FUNCTION_BLOCK ScrollFS_PHYS_Button (* Scroll list — accepts a single ScrollFull_S struct (geometry + physical controls), reads 6 on-screen Buttons and the direct-position input field, drives ScrollFS internally *)
  (* Standard: ISO 11783-6; Description: Copyright (c) 2026 Meisterschulen am Ostbahnhof This program and the accompanying materials are made available under the terms of the Eclipse Public License 2.0 which is available at https://www.eclipse.org/legal/epl-2.0/ SPDX-License-Identifier: EPL-2.0 Same as ScrollFS_PHYS, but reads the 6 scroll controls as on-screen Button objects (Button_IE, listening for BT_PRESSED_LATCHED) instead of physical SoftKeys — for masks where scrolling is operated via touch/on-screen buttons rather than the SoftKey column. Reuses the same ScrollFull_S / ScrollControls_S structs (the 6 IDs just point at Button objects instead of Key objects) and the same internal ScrollFS position engine. See Workspace_Scroll/SCROLL_KONZEPT.md for the full derivation. *)
  (* Version 1.1, 2026-09-05, Franz Höpfinger, Meisterschulen am Ostbahnhof, Add xScale flag, passed through to the internal ScrollFS *)
  (* Version 1.0, 2026-08-09, Franz Höpfinger, Meisterschulen am Ostbahnhof, initial API and implementation and/or initial documentation *)
  PACKAGE isobus::UT::Q;
  IMPORT isobus::utils::scroll::ScrollFull_S;
  IMPORT isobus::UT::Q::ScrollFS;
  IMPORT iec61131::selection::F_MOVE;
  IMPORT iec61131::conversion::F_DWORD_TO_DINT;
  IMPORT isobus::UT::io::Button::Button_IE;
  IMPORT isobus::UT::io::Button::ButtonActivationCode::BT_PRESSED_LATCHED;
  IMPORT isobus::UT::io::NumericValue::NumericValue_ID;
  IMPORT isobus::UT::Q::Q_NumericValue;
  IMPORT isobus::UT::Q::const::IDs::ID_NULL;
  IMPORT iec61131::selection::F_SEL;
  IMPORT iec61131::conversion::F_UINT_TO_UDINT;
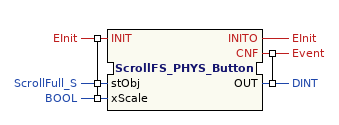
  EVENT_INPUT
    INIT : EInit WITH stObj, xScale; (* Service Initialization *)
  END_EVENT
  EVENT_OUTPUT
    INITO : EInit; (* Initialization Confirm *)
    CNF WITH OUT; (* Confirmation of a position change *)
  END_EVENT
  VAR_INPUT
    stObj : isobus::utils::scroll::ScrollFull_S; (* Complete scroll list configuration (geometry + operator controls), snapshotted at INIT *)
    xScale : BOOL := FALSE; (* FALSE (default) = bypass. TRUE = scale by the DM/SKM factor. Passed straight through to the internal ScrollFS instance. *)
  END_VAR
  VAR_OUTPUT
    OUT : DINT; (* Current scroll position (0..stObj.stGeometry.i32PosMax, in rows) *)
  END_VAR
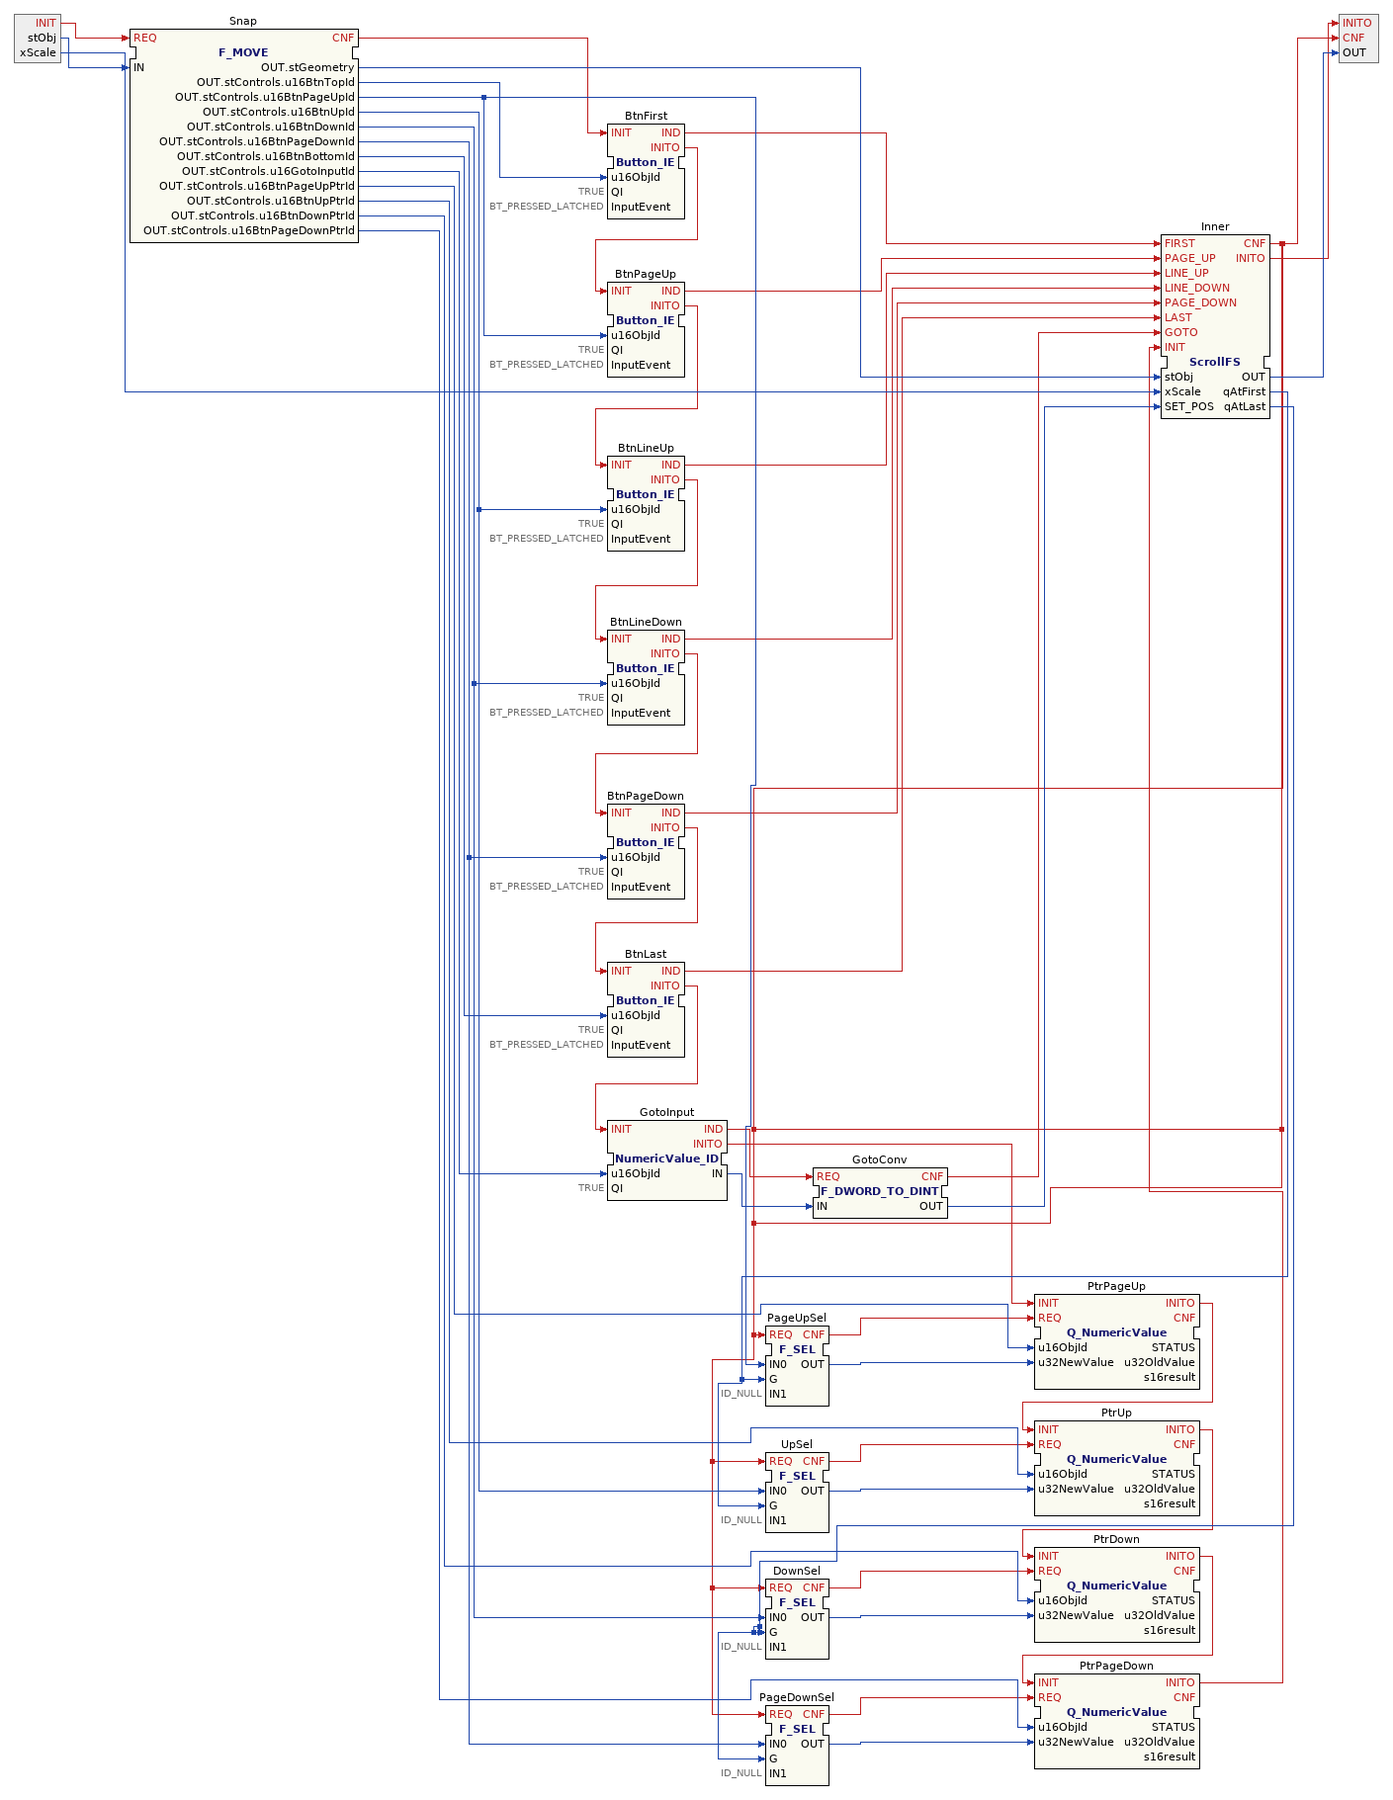
  FBS
    Snap : iec61131::selection::F_MOVE; {SET_ATTRIBUTE(DataType, isobus::utils::scroll::ScrollFull_S)}
    Inner : isobus::UT::Q::ScrollFS;
    BtnFirst : isobus::UT::io::Button::Button_IE(QI := TRUE, InputEvent := BT_PRESSED_LATCHED);
    BtnPageUp : isobus::UT::io::Button::Button_IE(QI := TRUE, InputEvent := BT_PRESSED_LATCHED);
    BtnLineUp : isobus::UT::io::Button::Button_IE(QI := TRUE, InputEvent := BT_PRESSED_LATCHED);
    BtnLineDown : isobus::UT::io::Button::Button_IE(QI := TRUE, InputEvent := BT_PRESSED_LATCHED);
    BtnPageDown : isobus::UT::io::Button::Button_IE(QI := TRUE, InputEvent := BT_PRESSED_LATCHED);
    BtnLast : isobus::UT::io::Button::Button_IE(QI := TRUE, InputEvent := BT_PRESSED_LATCHED);
    GotoInput : isobus::UT::io::NumericValue::NumericValue_ID(QI := TRUE);
    GotoConv : iec61131::conversion::F_DWORD_TO_DINT;
    PageUpSel : iec61131::selection::F_SEL(IN1 := ID_NULL);
    PtrPageUp : isobus::UT::Q::Q_NumericValue;
    UpSel : iec61131::selection::F_SEL(IN1 := ID_NULL);
    PtrUp : isobus::UT::Q::Q_NumericValue;
    DownSel : iec61131::selection::F_SEL(IN1 := ID_NULL);
    PtrDown : isobus::UT::Q::Q_NumericValue;
    PageDownSel : iec61131::selection::F_SEL(IN1 := ID_NULL);
    PtrPageDown : isobus::UT::Q::Q_NumericValue;
  END_FBS
  EVENT_CONNECTIONS
    INIT TO Snap.REQ;
    BtnFirst.IND TO Inner.FIRST;
    BtnPageUp.IND TO Inner.PAGE_UP;
    BtnLineUp.IND TO Inner.LINE_UP;
    BtnLineDown.IND TO Inner.LINE_DOWN;
    BtnPageDown.IND TO Inner.PAGE_DOWN;
    BtnLast.IND TO Inner.LAST;
    GotoInput.IND TO GotoConv.REQ;
    GotoConv.CNF TO Inner.GOTO;
    Inner.CNF TO CNF;
    Snap.CNF TO BtnFirst.INIT;
    BtnFirst.INITO TO BtnPageUp.INIT;
    BtnPageUp.INITO TO BtnLineUp.INIT;
    BtnLineUp.INITO TO BtnLineDown.INIT;
    BtnLineDown.INITO TO BtnPageDown.INIT;
    BtnPageDown.INITO TO BtnLast.INIT;
    BtnLast.INITO TO GotoInput.INIT;
    GotoInput.INITO TO PtrPageUp.INIT;
    PtrPageUp.INITO TO PtrUp.INIT;
    PtrUp.INITO TO PtrDown.INIT;
    PtrDown.INITO TO PtrPageDown.INIT;
    PtrPageDown.INITO TO Inner.INIT;
    Inner.INITO TO INITO;
    Inner.CNF TO PageUpSel.REQ;
    PageUpSel.CNF TO PtrPageUp.REQ;
    Inner.CNF TO UpSel.REQ;
    UpSel.CNF TO PtrUp.REQ;
    Inner.CNF TO DownSel.REQ;
    DownSel.CNF TO PtrDown.REQ;
    Inner.CNF TO PageDownSel.REQ;
    PageDownSel.CNF TO PtrPageDown.REQ;
  END_CONNECTIONS
  DATA_CONNECTIONS
    stObj TO Snap.IN;
    Snap.OUT.stGeometry TO Inner.stObj;
    xScale TO Inner.xScale;
    Snap.OUT.stControls.u16BtnTopId TO BtnFirst.u16ObjId;
    Snap.OUT.stControls.u16BtnPageUpId TO BtnPageUp.u16ObjId;
    Snap.OUT.stControls.u16BtnUpId TO BtnLineUp.u16ObjId;
    Snap.OUT.stControls.u16BtnDownId TO BtnLineDown.u16ObjId;
    Snap.OUT.stControls.u16BtnPageDownId TO BtnPageDown.u16ObjId;
    Snap.OUT.stControls.u16BtnBottomId TO BtnLast.u16ObjId;
    Snap.OUT.stControls.u16GotoInputId TO GotoInput.u16ObjId;
    GotoInput.IN TO GotoConv.IN;
    GotoConv.OUT TO Inner.SET_POS;
    Inner.OUT TO OUT;
    Snap.OUT.stControls.u16BtnPageUpPtrId TO PtrPageUp.u16ObjId;
    Snap.OUT.stControls.u16BtnPageUpId TO PageUpSel.IN0;
    Inner.qAtFirst TO PageUpSel.G;
    PageUpSel.OUT TO PtrPageUp.u32NewValue;
    Snap.OUT.stControls.u16BtnUpPtrId TO PtrUp.u16ObjId;
    Snap.OUT.stControls.u16BtnUpId TO UpSel.IN0;
    Inner.qAtFirst TO UpSel.G;
    UpSel.OUT TO PtrUp.u32NewValue;
    Snap.OUT.stControls.u16BtnDownPtrId TO PtrDown.u16ObjId;
    Snap.OUT.stControls.u16BtnDownId TO DownSel.IN0;
    Inner.qAtLast TO DownSel.G;
    DownSel.OUT TO PtrDown.u32NewValue;
    Snap.OUT.stControls.u16BtnPageDownPtrId TO PtrPageDown.u16ObjId;
    Snap.OUT.stControls.u16BtnPageDownId TO PageDownSel.IN0;
    Inner.qAtLast TO PageDownSel.G;
    PageDownSel.OUT TO PtrPageDown.u32NewValue;
  END_CONNECTIONS
END_FUNCTION_BLOCK
